{attribute 'pack_mode' := '1'}
TYPE ResultadoCiclo :
STRUCT
	producto  : STRING[25];
	OT:STRING[25];
	ciclo: INT;
	horaInicio: DT;
	horaFin: DT;
	retrasoPuesto: ARRAY[1..18] OF INT;
	tiempoPass: ARRAY[1..18] OF INT;
END_STRUCT
END_TYPE

(* stored: Version 1.1.0.1, ProductVersion 3.1.4024.12
   DUT ResultadoCiclo: Id {6de0a3f1-dd98-486b-a8cb-9e08ee304487} *)
